FUNCTION_BLOCK T_CartesianRobotModule EXTENDS FB_PackML_BaseModule
VAR
	_xAxis, _yAxis, _zAxis : I_Axis;
	_gripper : I_Gripper;
	_cartesianRobot : I_CartesianRobot;
	
	xAxisComponent : T_AxisComponent;
	yAxisComponent : T_AxisComponent;
	zAxisComponent : T_AxisComponent;
	gripperModule : T_GripperModule;
	
	productionMode : T_CartesianRobotProductionMode;
	maintenanceMode : T_CartesianRobotMaintenanceMode;
	manualMode : T_CartesianRobotManualMode;
END_VAR

METHOD GenericInitialise
VAR
	CartesianRobot : I_CartesianRobot;
	xAxis, yAxis, zAxis : I_Axis; 
	Gripper : I_Gripper;
	Cylinder : I_Cylinder;
END_VAR
_xAxis := xAxis;
_yAxis := yAxis;
_zAxis := zAxis;
_gripper := Gripper;
_cartesianRobot := CartesianRobot;

xAxisComponent.GenericInitialise(_xAxis);
yAxisComponent.GenericInitialise(_yAxis);
zAxisComponent.GenericInitialise(_zAxis);
gripperModule.GenericInitialise(gripper, Cylinder);

_cartesianRobot.GenericInitialise(xAxis, yAxis, zAxis, gripper);
productionMode.Initialise(THIS^);
maintenanceMode.Initialise(THIS^);
manualMode.Initialise(THIS^);

ComponentsCollection.AddComponent(xAxisComponent);
ComponentsCollection.AddComponent(yAxisComponent);
ComponentsCollection.AddComponent(zAxisComponent);
SubModulesCollection.AddModule(gripperModule);
END_METHOD

END_FUNCTION_BLOCK

(* stored: Version 1.1.0.1, ProductVersion 3.1.4024.12
   POU T_CartesianRobotModule: Id {7dc470ce-6b17-4384-bc6b-26e8ed9f37bb}, SpecialFunc None
   Method GenericInitialise: Id {9ab1df33-01ad-48c7-98d6-eb483ef184bd} *)
